FUNCTION_BLOCK CallButton (* Composite Function Block Type *)
  (* Standard: 61499-2 *)
  (* Version 0.0, 6/3/2016, Andrei, nxtControl GmbH, template *)
  PACKAGE Main;
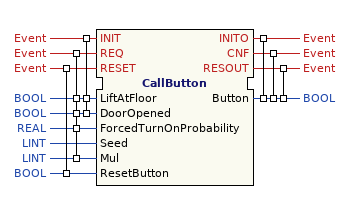
  EVENT_INPUT
    INIT WITH LiftAtFloor, DoorOpened; (* Initialization Request *)
    REQ WITH LiftAtFloor, DoorOpened, ForcedTurnOnProbability, Mul; (* Normal Execution Request *)
    RESET WITH ResetButton;
  END_EVENT
  EVENT_OUTPUT
    INITO WITH Button; (* Initialization Confirm *)
    CNF WITH Button; (* Execution Confirmation *)
    RESOUT WITH Button;
  END_EVENT
  VAR_INPUT
    LiftAtFloor : BOOL; (* Input event qualifier *)
    DoorOpened : BOOL;
    ForcedTurnOnProbability : REAL;
    Seed : LINT;
    Mul : LINT;
    ResetButton : BOOL;
  END_VAR
  VAR_OUTPUT
    Button : BOOL; (* Output event qualifier *)
  END_VAR
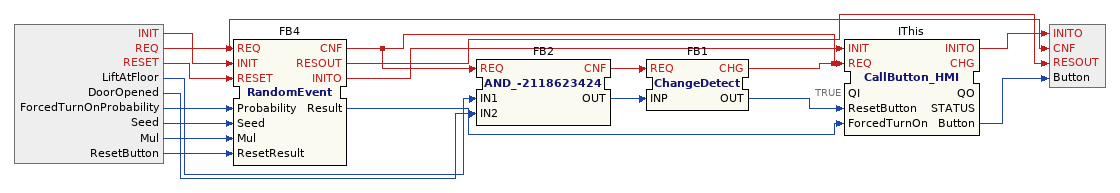
  FBS
    FB2 : AND_-2118623424; {SET_ATTRIBUTE(Configuration.GenericFBType.InterfaceParams, Runtime.Standard#CNT:=2;OUT:BOOL)}
    IThis : CallButton_HMI(QI := TRUE);
    FB4 : RandomEvent;
    FB1 : ChangeDetect;
  END_FBS
  EVENT_CONNECTIONS
    FB2.CNF TO FB1.REQ;
    REQ TO FB4.REQ;
    INIT TO FB4.INIT;
    FB4.CNF TO FB2.REQ;
    REQ TO CNF;
    RESET TO FB4.RESET;
    FB4.RESOUT TO RESOUT;
    FB4.INITO TO IThis.INIT;
    FB1.CHG TO IThis.REQ;
    FB4.CNF TO IThis.REQ;
    IThis.INITO TO INITO;
  END_CONNECTIONS
  DATA_CONNECTIONS
    LiftAtFloor TO FB2.IN1;
    DoorOpened TO FB2.IN2;
    FB2.OUT TO FB1.INP;
    ForcedTurnOnProbability TO FB4.Probability;
    Seed TO FB4.Seed;
    Mul TO FB4.Mul;
    ResetButton TO FB4.ResetResult;
    FB1.OUT TO IThis.ResetButton;
    FB4.Result TO IThis.ForcedTurnOn;
    IThis.Button TO Button;
  END_CONNECTIONS
END_FUNCTION_BLOCK
